TYPE ST_BisscEncoder :
STRUCT
	// Inclusive limits on encoder position (checks for values exceeding this inclusive range)
	// These values are just guesses - no units yet - no actual data - CHANGE BEFORE USE
	ncLLimit :	ULINT := 0;
	ncULimit :	ULINT := 100;
	// Readback for linear encoder's position
	encLoc	AT %I*	:	ULINT;
END_STRUCT
END_TYPE

(* stored: Version 1.1.0.1, ProductVersion 3.1.4020.12
   DUT ST_BisscEncoder: Id {ad70da24-7633-4882-90e5-890d60634d56} *)
